FUNCTION_BLOCK fbContext EXTENDS TcoCore.TcoContext
VAR
	
END_VAR

METHOD PROTECTED  Main
END_METHOD

END_FUNCTION_BLOCK

(* stored: Version 1.1.0.1, ProductVersion 3.1.4024.6
   POU fbContext: Id {d233a5a2-db40-465e-a632-646d6d0f5be7}, SpecialFunc None
   Method Main: Id {a8a64ca8-4dd3-4467-8956-c3b678a22f7c} *)
